ABB RobotStudio station: Lab_robotica_g6_cilindro.rsstn

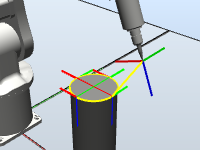
Station Solution98 (saved by RobotStudio 6.6.7701.1025)
Controller IRB_120_3kg_0.58m_1
  mechanical unit ROB_1: IRB120_3_58__01, 6 joints, base frame (0, 0, 0) mm
Layout (positions relative to the parent item):
  - IRB120_3_58__01 [mechanism, from Robots\IRB120_3_58_G_01.rslib] at (0, 0, 0) mm; joint values [0, 0, 0, 0, 0.5236, 0] (rad or m)
  - MyTool [mechanism, from Training Objects\myTool.rslib] at (364.35, 0, 594) mm, rotated rx 180 ry 60 rz 180 deg
  - Pieza_1 [part] at (-35.9, -51.66, 178.53) mm
Attachment: MyTool is attached to IRB120_3_58__01 / Link6
Attachment: Workobject_1 is attached to Pieza_1
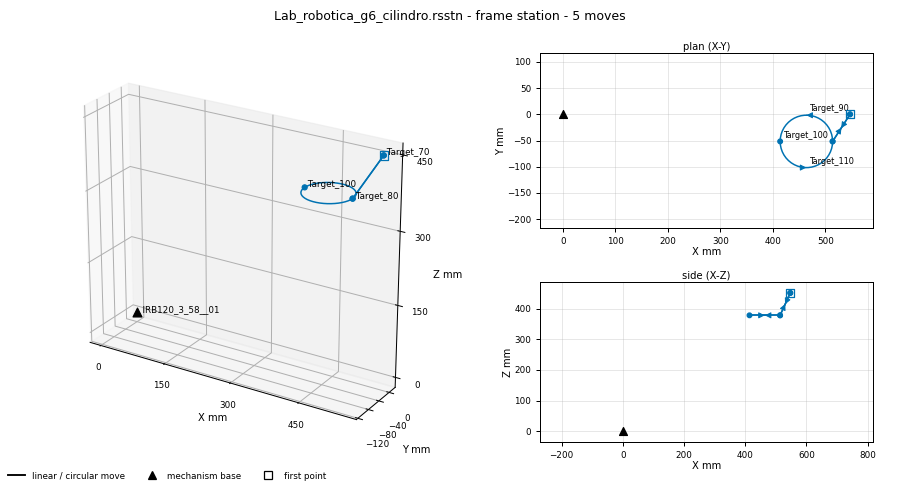
[picture p0: tool path of Lab_robotica_g6_cilindro.rsstn in frame station, 5 of 5 moves have a stored position in this frame; points joined in program order, loops and branches not executed]
Targets, tools, work objects and paths stored in the station, written as RAPID:
! task T_ROB1
MODULE CalibData
  PERS tooldata MyTool:=[TRUE,[[31.792631019,0,229.638935148],[0.945518576,0,0.325568154,0]],[1,[0,0,1],[1,0,0,0],0,0,0]];
  TASK PERS wobjdata Workobject_1:=[FALSE,TRUE,"",[[-35.90378533,-51.664067408,178.525901642],[1,0,0,0]],[[0,0,0],[1,0,0,0]]];
ENDMODULE

! task T_ROB1
MODULE Module1
  CONST robtarget Target_10:=[[500,0,200],[0,0,1,0],[0,0,0,0],[9E+09,9E+09,9E+09,9E+09,9E+09,9E+09]];
  CONST robtarget Target_70:=[[547.33065187,0,451.647288113],[0.19080896,0,0.98162719,0],[0,0,0,0],[9E+09,9E+09,9E+09,9E+09,9E+09,9E+09]];
  CONST robtarget Target_80:=[[550,0,200],[0,0,1,0],[0,0,0,0],[9E+09,9E+09,9E+09,9E+09,9E+09,9E+09]];
  CONST robtarget Target_90:=[[500,50,200],[0,0,1,0],[0,0,0,0],[9E+09,9E+09,9E+09,9E+09,9E+09,9E+09]];
  CONST robtarget Target_100:=[[450,0,200],[0,0,1,0],[0,0,0,0],[9E+09,9E+09,9E+09,9E+09,9E+09,9E+09]];
  CONST robtarget Target_110:=[[500,-50,200],[0,0,1,0],[0,0,0,0],[9E+09,9E+09,9E+09,9E+09,9E+09,9E+09]];
  CONST robtarget Target_120:=[[550,0,200],[0,0,1,0],[0,0,0,0],[9E+09,9E+09,9E+09,9E+09,9E+09,9E+09]];
  PROC Path_10()
    MoveL Target_70,v20,fine,MyTool\WObj:=wobj0;
    MoveL Target_80,v20,fine,MyTool\WObj:=Workobject_1;
    MoveC Target_90,Target_100,v20,fine,MyTool\WObj:=Workobject_1;
    MoveC Target_110,Target_120,v20,fine,MyTool\WObj:=Workobject_1;
    MoveL Target_70,v20,fine,MyTool\WObj:=wobj0;
  ENDPROC
ENDMODULE

